// Collection that exposes only immutable methods and properties of a collection that implements I_Set.
{attribute 'enable_dynamic_creation'}
FUNCTION_BLOCK FB_Immutable_Set IMPLEMENTS I_Immutable_Set
VAR_INPUT
	ipSet : I_Set;
END_VAR
VAR_STAT
	fbDefault_Immutable_List : FB_Immutable_List;
END_VAR

// Number of items in the collection.
PROPERTY _Count : T_Capacity
GET
IF THIS^.ipSet = 0 THEN RETURN; END_IF
	
_Count := THIS^.ipSet._Count;
END_GET
END_PROPERTY

// Checks if collection is empty.
PROPERTY _Empty : BOOL
GET
IF THIS^.ipSet = 0 THEN _Empty := TRUE; RETURN; END_IF
	
_Empty := THIS^.ipSet._Empty;
END_GET
END_PROPERTY

// Error status of the collection.
PROPERTY _Error_Status : T_Error
GET
IF THIS^.ipSet = 0 THEN 
	_Error_Status := F_Error(TRUE, GVL_Errors.ERR_INVALID_INTERFACE, 'The interface ipSet is null.');
	RETURN; 
	END_IF
	
_Error_Status := THIS^.ipSet._Error_Status;
END_GET
END_PROPERTY

// Checks if item is contained in set.
METHOD Contains : BOOL
VAR_INPUT
	Item : ANY; // Item to find.
END_VAR
IF THIS^.ipSet = 0 THEN RETURN; END_IF

Contains := THIS^.ipSet.Contains(Item);
END_METHOD

// Gets an immutable list of the values in the set.
METHOD Get_Values : I_Immutable_List
VAR
END_VAR
IF THIS^.ipSet = 0 THEN 
	Get_Values := THIS^.fbDefault_Immutable_List;
	RETURN; 
	END_IF

Get_Values := THIS^.ipSet.Get_Values();
END_METHOD

END_FUNCTION_BLOCK

(* stored: Version 1.1.0.1
   POU FB_Immutable_Set: Id {3afbf122-9852-03b8-0749-44fef68dc495}, SpecialFunc None
   Property _Count: Id {e75b6bd0-00bf-09b5-1d1e-a52e85bd879c}
   Get Get: Id {a56c62de-8d3e-0a63-3194-38dcd920b3f8}
   Property _Empty: Id {18c8bc00-2436-0ecf-1c24-280bdd534b78}
   Get Get: Id {5efbca70-23d1-0763-0668-ce9270860e37}
   Property _Error_Status: Id {7c517ed0-6a3a-0c83-0d5f-3b2057631059}
   Get Get: Id {05634e8b-9183-076a-0814-958c108bb693}
   Method Contains: Id {a4babfbd-b0c3-0e0f-37a7-97164cd0541d}
   Method Get_Values: Id {7932ed8d-68b8-08c1-17c4-535dddfe387d} *)
